FUNCTION AsTagged : Result
VAR_INPUT
	iSource	: I_Component;
END_VAR
VAR_OUTPUT
	iDest	: I_Tagged;
END_VAR

IF iSource = 0 THEN
	AsTagged := Err.Itf0;
	RETURN;
END_IF

IF __QUERYINTERFACE(iSource, iDest) THEN
	AsTagged := Ok;
ELSE
	AsTagged := Err.NoMatch;
END_IF

END_FUNCTION

(* stored: Version 1.1.0.1
   POU AsTagged: Id {037a1bf0-02fe-469d-a7f0-fdd83b19b2c8}, SpecialFunc None *)
